VAR_GLOBAL // STATE
    p_x: DINT;
    p_t: LREAL;
END_VAR

(* stored: ProductVersion 3.1.0.18, Version 1.1.0.1 *)
